FUNCTION F_MaxReportTime_TO_Time : TIME
VAR_INPUT
	sTimeIn : STRING;
END_VAR
VAR
	TempOT : OTSTRUCT;
	
	
END_VAR

//'12:34:56:789';
TempOT.wHour			:= STRING_TO_WORD(LEFT(sTimeIn,2));
TempOT.wMinute			:= STRING_TO_WORD(MID(sTimeIn,2,4));
TempOT.wSecond			:= STRING_TO_WORD(MID(sTimeIn,2,7));

F_MaxReportTime_TO_Time	:= OTSTRUCT_TO_TIME(OTIN:= TempOT);

END_FUNCTION

(* stored: Version 1.1.0.1, ProductVersion 3.1.4020.6
   POU F_MaxReportTime_TO_Time: Id {f2a996e7-3f4e-4bba-8d94-ff8c17360b78}, SpecialFunc None *)
